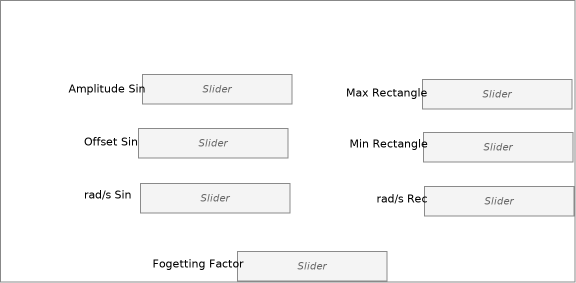
VISUALIZATION Visualization  // 576x283
    Slider (142,74 150x30), variable: MAIN.r_AmplitudeSin, scale 0..50
    Label (32,74 150x30), "Amplitude Sin"
    Slider (422,79 150x30), variable: MAIN.r_MaxValueRec, scale 0..50
    Label (312,78 150x30), "Max Rectangle"
    Slider (423,132 150x30), variable: MAIN.r_MinValueRec, scale -50..0
    Label (314,129 150x30), "Min Rectangle"
    Slider (140,183 150x30), variable: MAIN.r_KreisfrequenzSin, scale 0..100
    Label (33,180 150x30), "rad/s Sin"
    Slider (424,186 150x30), variable: MAIN.r_KreisfrequenzRec, scale 0..100
    Label (327,184 150x30), "rad/s Rec"
    Slider (138,128 150x30), variable: MAIN.r_OffsetSin, scale -20..20
    Label (36,127 150x30), "Offset Sin"
    Slider (237,251 150x30), variable: MAIN.r_FogettingFactor, scale 0..0.999
    Label (123,249 150x30), "Fogetting Factor"
END_VISUALIZATION

(* stored: Version 1.1.0.1, ProductVersion 3.1.4022.12
   Visu Visualization: Id {69a786f7-1e91-4d1f-ae36-e0d3c162118d} *)
